Staubli VAL3: simulation.pgx

program simulation()
  local string l_sMessage
begin
  //
  // SIMULATION
  //
  // syncro
  bLarge=true
  use:nPage=200
  watch(cycleStatus:pCycleProg.sID!="",1)
  use:bUseRefresh=true
  cls()
  do
    nKey=getKey()
    // REFRESH
    if cycleStatus:bSimulation
      call refresh()
    endIf
    call use:type(31,13,"STOP ")
    // look for the restart button
    if cycleStatus:bPause
      call use:type(23,13,"RESTART")
      if nKey==276
        call OnEvent:resumeCycle()
      endIf
    else
      call use:type(23,13,"        ")
    endIf
    delay(0)
  until nKey==255 or nKey==277 or cycleStatus:bToStop or cycleStatus:bSimulation==false
  //
  if nKey==255 or nKey==277
    cycleStatus:bToStop=true
    watch(cycleStatus:bToStop==false,1)
  endIf
  // leave
  call use:nullKey(nKey)
end
